TYPE ST_DIAGNOSTICMESSAGE :
STRUCT
    stDiagnosticCode : ST_DIAGNOSTICCODE;
    stFlags : ST_FLAGS;
    nTextIdentityReferenceToESIFile : UINT;
    sTimeStamp : STRING(29);
END_STRUCT
END_TYPE

(* stored: Version 1.1.0.1
   DUT ST_DIAGNOSTICMESSAGE: Id {b78917fa-7725-4496-a05b-ea21f85e2a59} *)
